TYPE TemperatureStructure :
STRUCT
	RoomTemperature : REAL;
	BathRoomTemperature : REAL;
	SomeOtherData : DINT;
	ekstra	: HaProduct;
END_STRUCT
END_TYPE

(* stored: Version 1.1.0.1, ProductVersion 3.1.4024.12
   DUT TemperatureStructure: Id {bdb6708b-dce7-4d63-abfa-3db6627c8b4a} *)
